(* PLC project static_torsion.project, CODESYS CODESYS V3.5 SP17 Patch 3 *)
(* stored: creationDateTime 1970-01-01T00:00:00, modificationDateTime 2026-06-22T15:12:39.4699931 *)

{attribute 'hasanytype'}
FUNCTION to_word_ : WORD
  VAR_INPUT
    {attribute 'anytypeclass' := 'ANY'}
    in : __SYSTEM.AnyType;
  END_VAR
  VAR
    p_word : POINTER TO WORD;
  END_VAR

            // Принимает на входе значение любого типа длиной 1 байт
// Возвращает значение типа WORD
p_word := in.pValue;	// Преобразуем указатель на BYTE в указатель на WORD
to_word_ := p_word^;
          
END_FUNCTION
